Staubli VAL3: JointForce.dtx

public num jf[6]
